// Writes a 64-bit little-endian integer.
FUNCTION F_WriteRawLittleEndian64 : HRESULT
VAR_IN_OUT      
    stCtx : ST_WriteContext;
END_VAR
VAR_INPUT CONSTANT
    nValue : ULINT;
END_VAR
VAR CONSTANT
    cLength : UDINT := SIZEOF(nValue);
END_VAR

F_WriteRawLittleEndian64 := F_WriteToBuffer(stCtx, F_ToAnyType(nValue), cLength);

END_FUNCTION

(* stored: Version 1.1.0.1
   POU F_WriteRawLittleEndian64: Id {b65dc470-e97e-4ecb-bd6d-af355d41c263}, SpecialFunc None *)
